{attribute 'GeneratedUsingTerminal: EP5101-0011-0016'}
{attribute addProperty BoxType "EP5101-0011-0016"}
{attribute addProperty Id "EtcSlaveTerminalBaseENC_Status_compactAT %I*ENC_Status_compact_7D3464F320ENC_Control_compactAT %Q*ENC_Control_compact_21E2D14D6WcStateAT %I*WcState_9091E0EB2InfoDataAT %I*InfoData_32EB74EA10"}
{attribute addProperty CRC "3997198820"}
{attribute addProperty Size "38"}
TYPE EP5101_EE4069E4 EXTENDS EtcSlaveTerminalBase :
STRUCT
	{attribute addProperty Name "ENC_Status_compact"}
	ENC_Status_compact : ENC_Status_compact_7D3464F3;
	{attribute addProperty Name "ENC_Control_compact"}
	ENC_Control_compact : ENC_Control_compact_21E2D14D;
	{attribute addProperty Name "WcState"}
	WcState : WcState_9091E0EB;
	{attribute addProperty Name "InfoData"}
	InfoData : InfoData_32EB74EA;
END_STRUCT
END_TYPE

(* stored: Version 1.2.0.0, ProductVersion 3.1.4024.9
   DUT EP5101_EE4069E4: Id {49dd4d51-c85e-4df7-80e8-52bb29a64a73} *)
